// TIA Portal V21 export
TYPE "coneCrusherSimHMI"
   STRUCT
      cmdWord : Word;
      ambientTemp : LReal;
   END_STRUCT;
END_TYPE
